// TIA Portal V20 export
TYPE "UDT_Service_ParaIndexInfoDigBin"
   STRUCT
      Index : Int;
      DisplayIndex : Int;
   END_STRUCT;
END_TYPE
